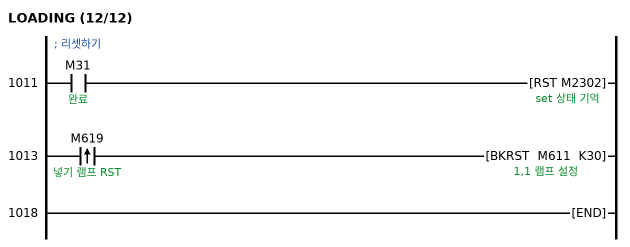
[picture p24: ladder of LOADING, rungs at steps 1011 to 1018]
; 리셋하기
1011  LD      M31  ; 완료
      RST     M2302  ; set 상태 기억
1013  LDP     M619  ; 넣기 램프 RST
      BKRST   M611 K30  ; 1,1 램프 설정
1018  END
END_PROGRAM

PROGRAM UNLOAD
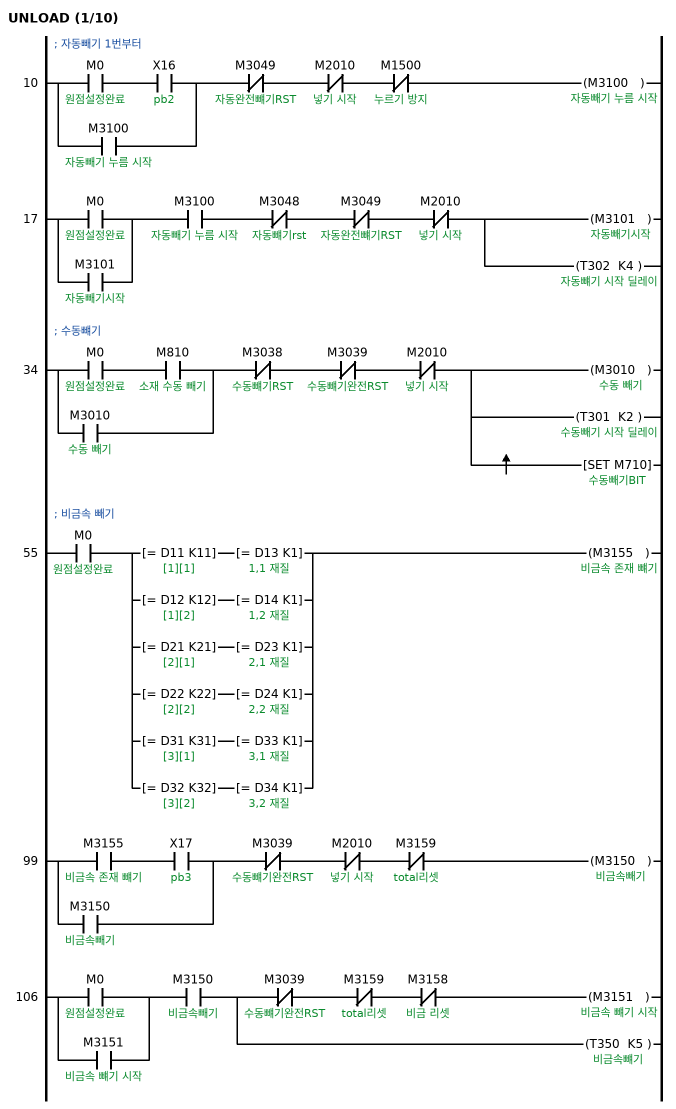
; 자동빼기 1번부터
10    LD      M0  ; 원점설정완료
      AND     X16  ; pb2
      OR      M3100  ; 자동빼기 누름 시작
      ANI     M3049  ; 자동완전뺴기RST
      ANI     M2010  ; 넣기 시작
      ANI     M1500  ; 누르기 방지
      OUT     M3100  ; 자동빼기 누름 시작
17    LD      M0  ; 원점설정완료
      OR      M3101  ; 자동빼기시작
      AND     M3100  ; 자동빼기 누름 시작
      ANI     M3048  ; 자동뺴기rst
      ANI     M3049  ; 자동완전뺴기RST
      ANI     M2010  ; 넣기 시작
      OUT     M3101  ; 자동빼기시작
      OUT     T302 K4  ; 자동뺴기 시작 딜레이
; 수동뺴기
34    LD      M0  ; 원점설정완료
      AND     M810  ; 소재 수동 빼기
      OR      M3010  ; 수동 빼기
      ANI     M3038  ; 수동뺴기RST
      ANI     M3039  ; 수동뺴기완전RST
      ANI     M2010  ; 넣기 시작
      OUT     M3010  ; 수동 빼기
      OUT     T301 K2  ; 수동빼기 시작 딜레이
      MEP
      SET     M710  ; 수동빼기BIT
; 비금속 빼기
55    LD      M0  ; 원점설정완료
      LD=     D11 K11  ; [1][1]
      AND=    D13 K1  ; 1,1 재질
      LD=     D12 K12  ; [1][2]
      AND=    D14 K1  ; 1,2 재질
      ORB
      LD=     D21 K21  ; [2][1]
      AND=    D23 K1  ; 2,1 재질
      ORB
      LD=     D22 K22  ; [2][2]
      AND=    D24 K1  ; 2,2 재질
      ORB
      LD=     D31 K31  ; [3][1]
      AND=    D33 K1  ; 3,1 재질
      ORB
      LD=     D32 K32  ; [3][2]
      AND=    D34 K1  ; 3,2 재질
      ORB
      ANB
      OUT     M3155  ; 비금속 존재 뺴기
99    LD      M3155  ; 비금속 존재 뺴기
      AND     X17  ; pb3
      OR      M3150  ; 비금속빼기
      ANI     M3039  ; 수동뺴기완전RST
      ANI     M2010  ; 넣기 시작
      ANI     M3159  ; total리셋
      OUT     M3150  ; 비금속빼기
106   LD      M0  ; 원점설정완료
      OR      M3151  ; 비금속 뺴기 시작
      AND     M3150  ; 비금속빼기
      MPS
      ANI     M3039  ; 수동뺴기완전RST
      ANI     M3159  ; total리셋
      ANI     M3158  ; 비금 리셋
      OUT     M3151  ; 비금속 뺴기 시작
      MPP
      OUT     T350 K5  ; 비금속뺴기
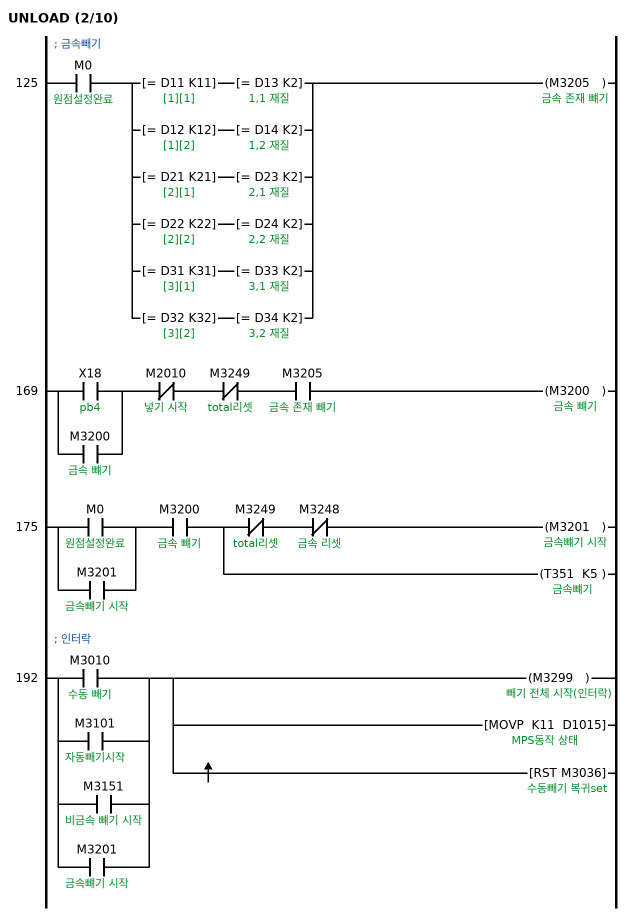
; 금속빼기
125   LD      M0  ; 원점설정완료
      LD=     D11 K11  ; [1][1]
      AND=    D13 K2  ; 1,1 재질
      LD=     D12 K12  ; [1][2]
      AND=    D14 K2  ; 1,2 재질
      ORB
      LD=     D21 K21  ; [2][1]
      AND=    D23 K2  ; 2,1 재질
      ORB
      LD=     D22 K22  ; [2][2]
      AND=    D24 K2  ; 2,2 재질
      ORB
      LD=     D31 K31  ; [3][1]
      AND=    D33 K2  ; 3,1 재질
      ORB
      LD=     D32 K32  ; [3][2]
      AND=    D34 K2  ; 3,2 재질
      ORB
      ANB
      OUT     M3205  ; 금속 존재 뺴기
169   LD      X18  ; pb4
      OR      M3200  ; 금속 뺴기
      ANI     M2010  ; 넣기 시작
      ANI     M3249  ; total리셋
      AND     M3205  ; 금속 존재 뺴기
      OUT     M3200  ; 금속 뺴기
175   LD      M0  ; 원점설정완료
      OR      M3201  ; 금속뺴기 시작
      AND     M3200  ; 금속 뺴기
      MPS
      ANI     M3249  ; total리셋
      ANI     M3248  ; 금속 리셋
      OUT     M3201  ; 금속뺴기 시작
      MPP
      OUT     T351 K5  ; 금속뺴기
; 인터락
192   LD      M3010  ; 수동 빼기
      OR      M3101  ; 자동빼기시작
      OR      M3151  ; 비금속 뺴기 시작
      OR      M3201  ; 금속뺴기 시작
      OUT     M3299  ; 빼기 전체 시작(인터락)
      MOVP    K11 D1015  ; MPS동작 상태
      MEP
      RST     M3036  ; 수동빼기 복귀set
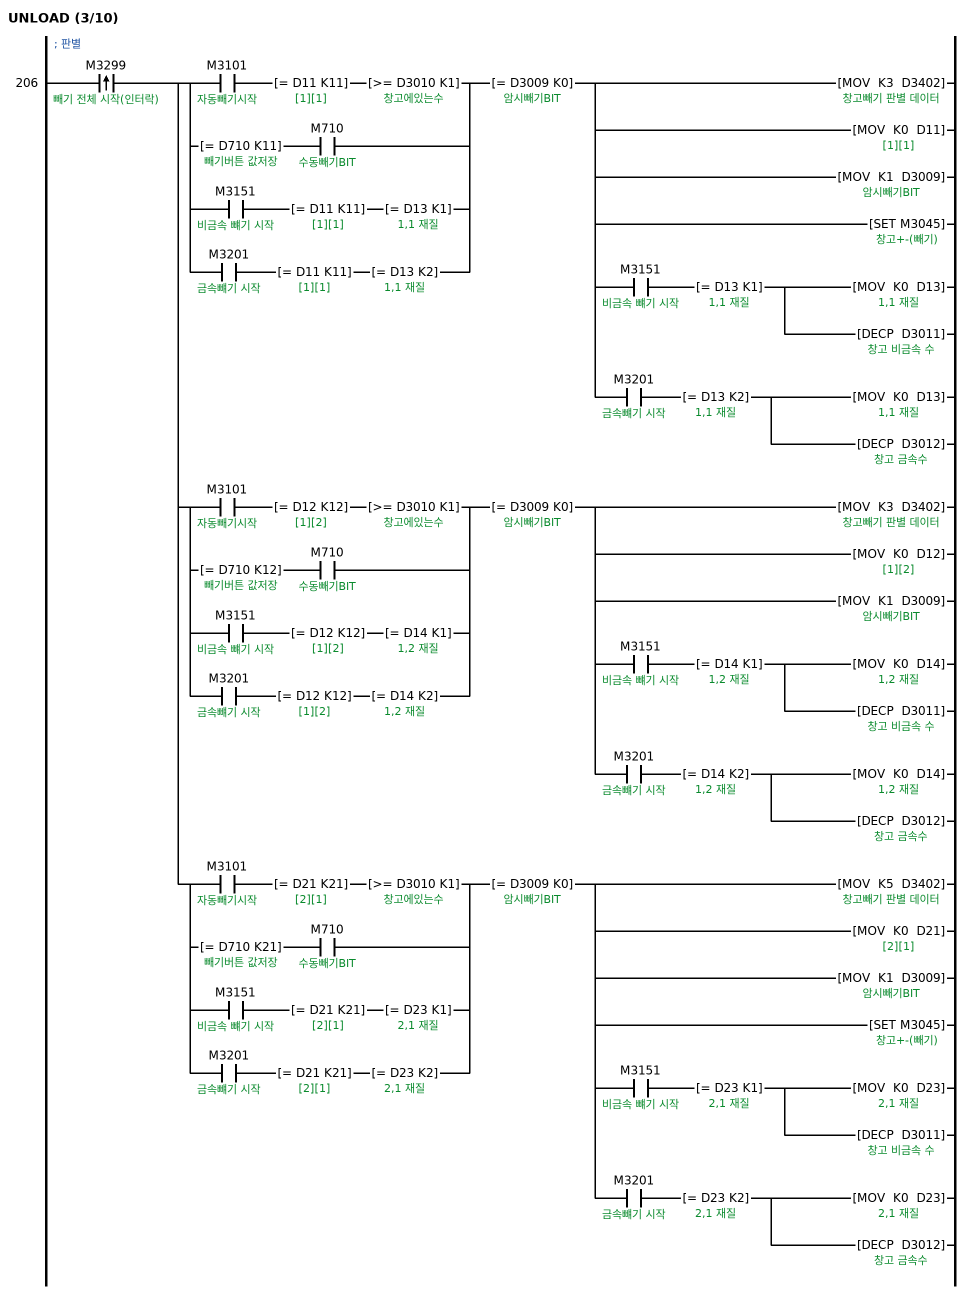
; 판별
206   LDP     M3299  ; 빼기 전체 시작(인터락)
      MPS
      LD      M3101  ; 자동빼기시작
      AND=    D11 K11  ; [1][1]
      AND>=   D3010 K1  ; 창고에있는수
      LD=     D710 K11  ; 빼기버튼 값저장
      AND     M710  ; 수동빼기BIT
      ORB
      LD      M3151  ; 비금속 뺴기 시작
      AND=    D11 K11  ; [1][1]
      AND=    D13 K1  ; 1,1 재질
      ORB
      LD      M3201  ; 금속뺴기 시작
      AND=    D11 K11  ; [1][1]
      AND=    D13 K2  ; 1,1 재질
      ORB
      ANB
      AND=    D3009 K0  ; 암시빼기BIT
      MOV     K3 D3402  ; 창고빼기 판별 데이터
      MOV     K0 D11
      MOV     K1 D3009
      SET     M3045  ; 창고+-(빼기)
      MPS
      AND     M3151  ; 비금속 뺴기 시작
      AND=    D13 K1  ; 1,1 재질
      MOV     K0 D13
      DECP    D3011  ; 창고 비금속 수
      MPP
      AND     M3201  ; 금속뺴기 시작
      AND=    D13 K2  ; 1,1 재질
      MOV     K0 D13
      DECP    D3012  ; 창고 금속수
      MRD
      LD      M3101  ; 자동빼기시작
      AND=    D12 K12  ; [1][2]
      AND>=   D3010 K1  ; 창고에있는수
      LD=     D710 K12  ; 빼기버튼 값저장
      AND     M710  ; 수동빼기BIT
      ORB
      LD      M3151  ; 비금속 뺴기 시작
      AND=    D12 K12  ; [1][2]
      AND=    D14 K1  ; 1,2 재질
      ORB
      LD      M3201  ; 금속뺴기 시작
      AND=    D12 K12  ; [1][2]
      AND=    D14 K2  ; 1,2 재질
      ORB
      ANB
      AND=    D3009 K0  ; 암시빼기BIT
      MOV     K3 D3402
      MOV     K0 D12
      MOV     K1 D3009
      MPS
      AND     M3151  ; 비금속 뺴기 시작
      AND=    D14 K1  ; 1,2 재질
      MOV     K0 D14
      DECP    D3011
      MPP
      AND     M3201  ; 금속뺴기 시작
      AND=    D14 K2  ; 1,2 재질
      MOV     K0 D14
      DECP    D3012
      MPP
      LD      M3101  ; 자동빼기시작
      AND=    D21 K21  ; [2][1]
      AND>=   D3010 K1  ; 창고에있는수
      LD=     D710 K21  ; 빼기버튼 값저장
      AND     M710  ; 수동빼기BIT
      ORB
      LD      M3151  ; 비금속 뺴기 시작
      AND=    D21 K21  ; [2][1]
      AND=    D23 K1  ; 2,1 재질
      ORB
      LD      M3201  ; 금속뺴기 시작
      AND=    D21 K21  ; [2][1]
      AND=    D23 K2  ; 2,1 재질
      ORB
      ANB
      AND=    D3009 K0  ; 암시빼기BIT
      MOV     K5 D3402
      MOV     K0 D21
      MOV     K1 D3009
      SET     M3045  ; 창고+-(빼기)
      MPS
      AND     M3151  ; 비금속 뺴기 시작
      AND=    D23 K1  ; 2,1 재질
      MOV     K0 D23
      DECP    D3011
      MPP
      AND     M3201  ; 금속뺴기 시작
      AND=    D23 K2  ; 2,1 재질
      MOV     K0 D23
      DECP    D3012
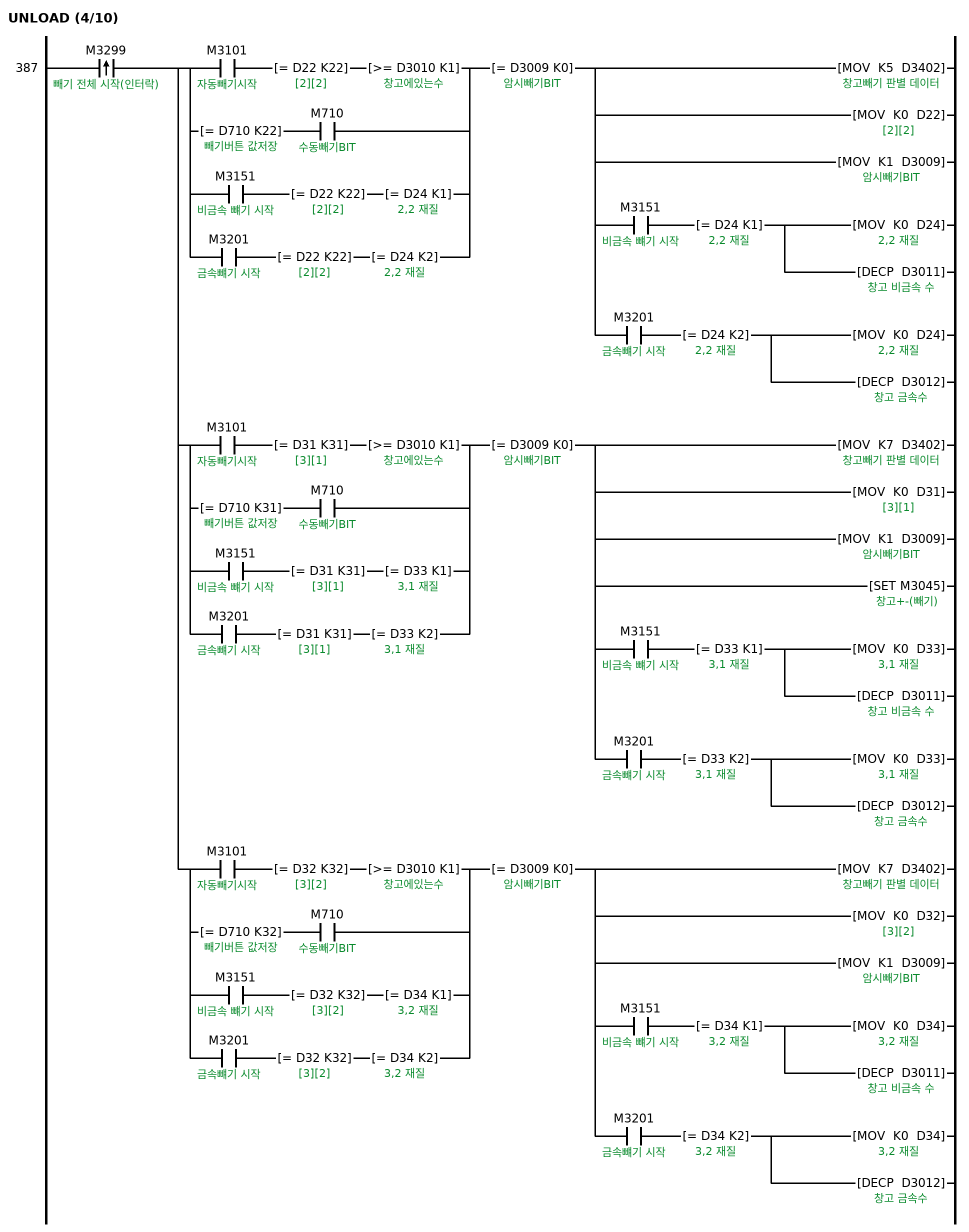
387   LDP     M3299  ; 빼기 전체 시작(인터락)
      MPS
      LD      M3101  ; 자동빼기시작
      AND=    D22 K22  ; [2][2]
      AND>=   D3010 K1  ; 창고에있는수
      LD=     D710 K22  ; 빼기버튼 값저장
      AND     M710  ; 수동빼기BIT
      ORB
      LD      M3151  ; 비금속 뺴기 시작
      AND=    D22 K22  ; [2][2]
      AND=    D24 K1  ; 2,2 재질
      ORB
      LD      M3201  ; 금속뺴기 시작
      AND=    D22 K22  ; [2][2]
      AND=    D24 K2  ; 2,2 재질
      ORB
      ANB
      AND=    D3009 K0  ; 암시빼기BIT
      MOV     K5 D3402
      MOV     K0 D22
      MOV     K1 D3009
      MPS
      AND     M3151  ; 비금속 뺴기 시작
      AND=    D24 K1  ; 2,2 재질
      MOV     K0 D24
      DECP    D3011
      MPP
      AND     M3201  ; 금속뺴기 시작
      AND=    D24 K2  ; 2,2 재질
      MOV     K0 D24
      DECP    D3012
      MRD
      LD      M3101  ; 자동빼기시작
      AND=    D31 K31  ; [3][1]
      AND>=   D3010 K1  ; 창고에있는수
      LD=     D710 K31  ; 빼기버튼 값저장
      AND     M710  ; 수동빼기BIT
      ORB
      LD      M3151  ; 비금속 뺴기 시작
      AND=    D31 K31  ; [3][1]
      AND=    D33 K1  ; 3,1 재질
      ORB
      LD      M3201  ; 금속뺴기 시작
      AND=    D31 K31  ; [3][1]
      AND=    D33 K2  ; 3,1 재질
      ORB
      ANB
      AND=    D3009 K0  ; 암시빼기BIT
      MOV     K7 D3402
      MOV     K0 D31
      MOV     K1 D3009
      SET     M3045  ; 창고+-(빼기)
      MPS
      AND     M3151  ; 비금속 뺴기 시작
      AND=    D33 K1  ; 3,1 재질
      MOV     K0 D33
      DECP    D3011
      MPP
      AND     M3201  ; 금속뺴기 시작
      AND=    D33 K2  ; 3,1 재질
      MOV     K0 D33
      DECP    D3012
      MPP
      LD      M3101  ; 자동빼기시작
      AND=    D32 K32  ; [3][2]
      AND>=   D3010 K1  ; 창고에있는수
      LD=     D710 K32  ; 빼기버튼 값저장
      AND     M710  ; 수동빼기BIT
      ORB
      LD      M3151  ; 비금속 뺴기 시작
      AND=    D32 K32  ; [3][2]
      AND=    D34 K1  ; 3,2 재질
      ORB
      LD      M3201  ; 금속뺴기 시작
      AND=    D32 K32  ; [3][2]
      AND=    D34 K2  ; 3,2 재질
      ORB
      ANB
      AND=    D3009 K0  ; 암시빼기BIT
      MOV     K7 D3402
      MOV     K0 D32
      MOV     K1 D3009
      MPS
      AND     M3151  ; 비금속 뺴기 시작
      AND=    D34 K1  ; 3,2 재질
      MOV     K0 D34
      DECP    D3011
      MPP
      AND     M3201  ; 금속뺴기 시작
      AND=    D34 K2  ; 3,2 재질
      MOV     K0 D34
      DECP    D3012
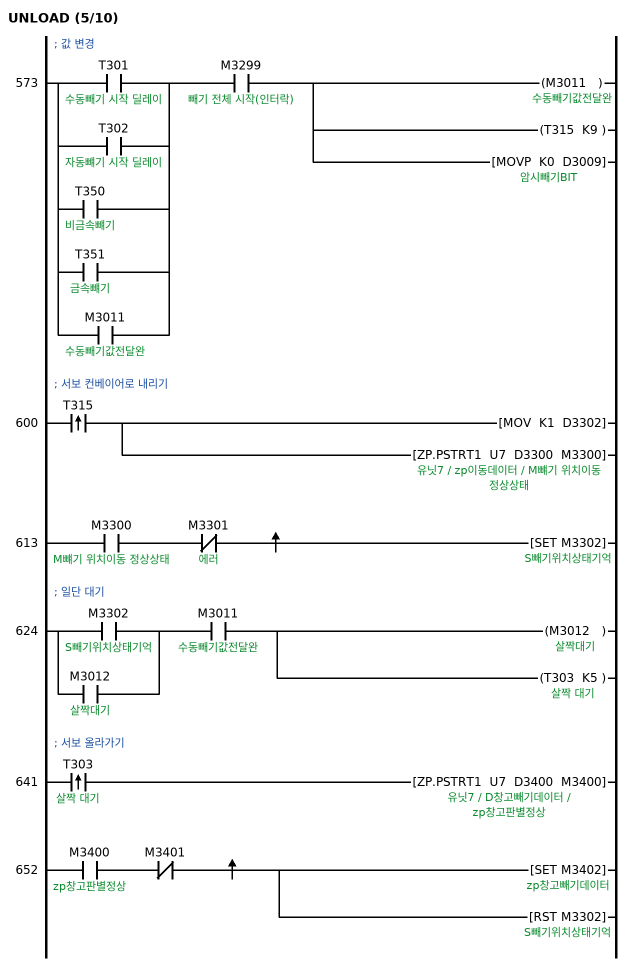
; 값 변경
573   LD      T301  ; 수동빼기 시작 딜레이
      OR      T302  ; 자동뺴기 시작 딜레이
      OR      T350  ; 비금속뺴기
      OR      T351  ; 금속뺴기
      OR      M3011  ; 수동빼기값전달완
      AND     M3299  ; 빼기 전체 시작(인터락)
      OUT     M3011  ; 수동빼기값전달완
      OUT     T315 K9
      MOVP    K0 D3009
; 서보 컨베이어로 내리기
600   LDP     T315
      MOV     K1 D3302
      ZP.PSTRT1 U7 D3300 M3300  ; 유닛7 / zp이동데이터 / M뺴기 위치이동 정상상태
613   LD      M3300  ; M뺴기 위치이동 정상상태
      ANI     M3301  ; 에러
      MEP
      SET     M3302  ; S빼기위치상태기억
; 일단 대기
624   LD      M3302  ; S빼기위치상태기억
      OR      M3012  ; 살짝대기
      AND     M3011  ; 수동빼기값전달완
      OUT     M3012  ; 살짝대기
      OUT     T303 K5  ; 살짝 대기
; 서보 올라가기
641   LDP     T303  ; 살짝 대기
      ZP.PSTRT1 U7 D3400 M3400  ; D창고빼기데이터 / zp창고판별정상
652   LD      M3400  ; zp창고판별정상
      ANI     M3401
      MEP
      SET     M3402  ; zp창고빼기데이터
      RST     M3302  ; S빼기위치상태기억
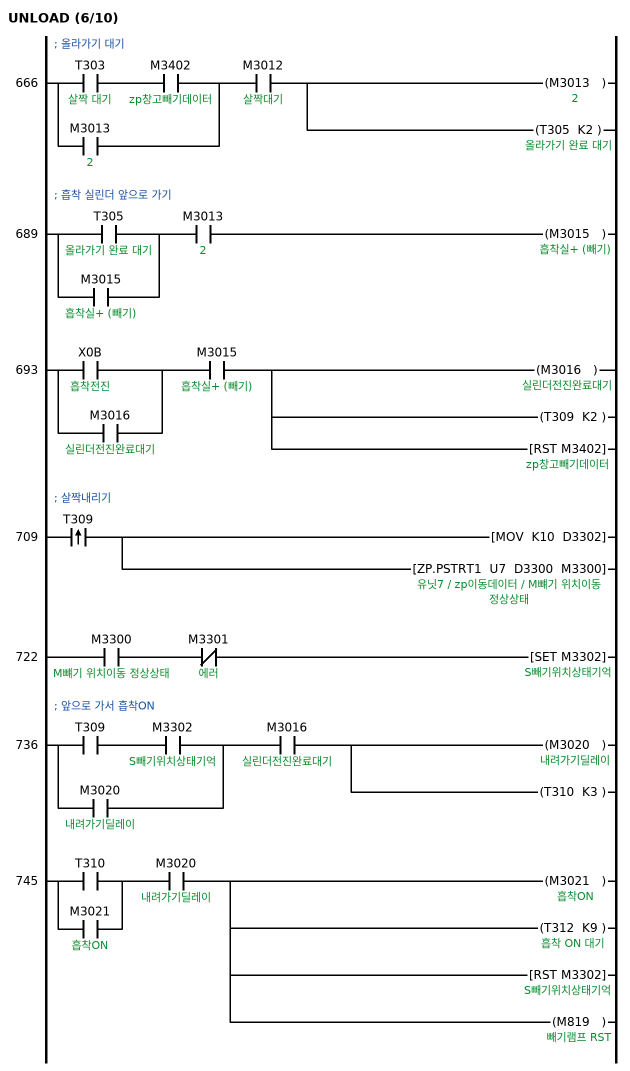
; 올라가기 대기
666   LD      T303  ; 살짝 대기
      AND     M3402  ; zp창고빼기데이터
      OR      M3013  ; 2
      AND     M3012  ; 살짝대기
      OUT     M3013  ; 2
      OUT     T305 K2  ; 올라가기 완료 대기
; 흡착 실린더 앞으로 가기
689   LD      T305  ; 올라가기 완료 대기
      OR      M3015  ; 흡착실+ (빼기)
      AND     M3013  ; 2
      OUT     M3015  ; 흡착실+ (빼기)
693   LD      X0B  ; 흡착전진
      OR      M3016  ; 실린더전진완료대기
      AND     M3015  ; 흡착실+ (빼기)
      OUT     M3016  ; 실린더전진완료대기
      OUT     T309 K2
      RST     M3402  ; zp창고빼기데이터
; 살짝내리기
709   LDP     T309
      MOV     K10 D3302
      ZP.PSTRT1 U7 D3300 M3300
722   LD      M3300  ; M뺴기 위치이동 정상상태
      ANI     M3301  ; 에러
      SET     M3302  ; S빼기위치상태기억
; 앞으로 가서 흡착ON
736   LD      T309
      AND     M3302  ; S빼기위치상태기억
      OR      M3020  ; 내려가기딜레이
      AND     M3016  ; 실린더전진완료대기
      OUT     M3020  ; 내려가기딜레이
      OUT     T310 K3
745   LD      T310
      OR      M3021  ; 흡착ON
      AND     M3020  ; 내려가기딜레이
      OUT     M3021  ; 흡착ON
      OUT     T312 K9  ; 흡착 ON 대기
      RST     M3302  ; S빼기위치상태기억
      OUT     M819  ; 빼기램프 RST
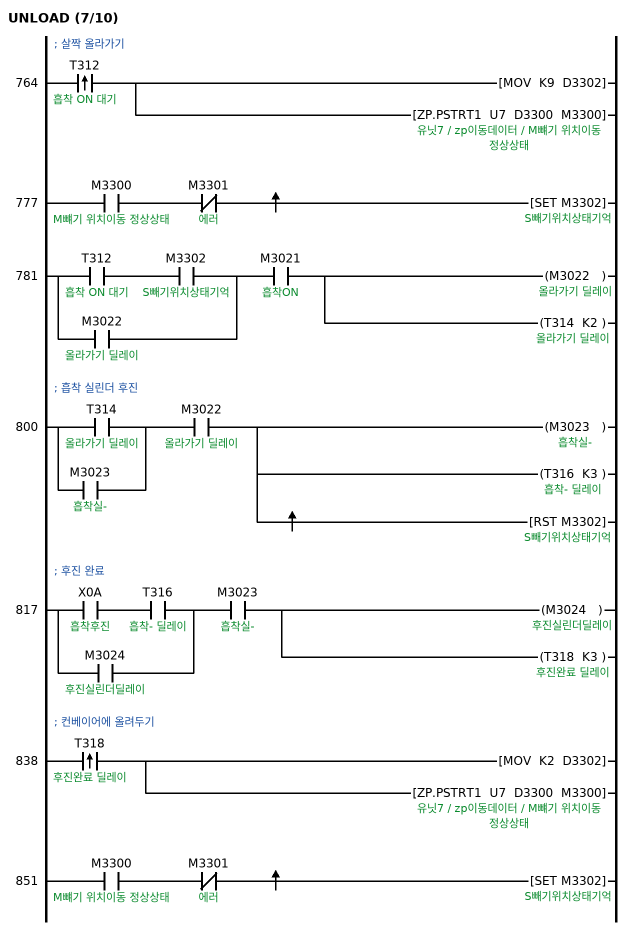
; 살짝 올라가기
764   LDP     T312  ; 흡착 ON 대기
      MOV     K9 D3302
      ZP.PSTRT1 U7 D3300 M3300
777   LD      M3300  ; M뺴기 위치이동 정상상태
      ANI     M3301  ; 에러
      MEP
      SET     M3302  ; S빼기위치상태기억
781   LD      T312  ; 흡착 ON 대기
      AND     M3302  ; S빼기위치상태기억
      OR      M3022  ; 올라가기 딜레이
      AND     M3021  ; 흡착ON
      OUT     M3022  ; 올라가기 딜레이
      OUT     T314 K2  ; 올라가기 딜레이
; 흡착 실린더 후진
800   LD      T314  ; 올라가기 딜레이
      OR      M3023  ; 흡착실-
      AND     M3022  ; 올라가기 딜레이
      OUT     M3023  ; 흡착실-
      OUT     T316 K3  ; 흡착- 딜레이
      MEP
      RST     M3302  ; S빼기위치상태기억
; 후진 완료
817   LD      X0A  ; 흡착후진
      AND     T316  ; 흡착- 딜레이
      OR      M3024  ; 후진실린더딜레이
      AND     M3023  ; 흡착실-
      OUT     M3024  ; 후진실린더딜레이
      OUT     T318 K3  ; 후진완료 딜레이
; 컨베이어에 올려두기
838   LDP     T318  ; 후진완료 딜레이
      MOV     K2 D3302
      ZP.PSTRT1 U7 D3300 M3300
851   LD      M3300  ; M뺴기 위치이동 정상상태
      ANI     M3301  ; 에러
      MEP
      SET     M3302  ; S빼기위치상태기억
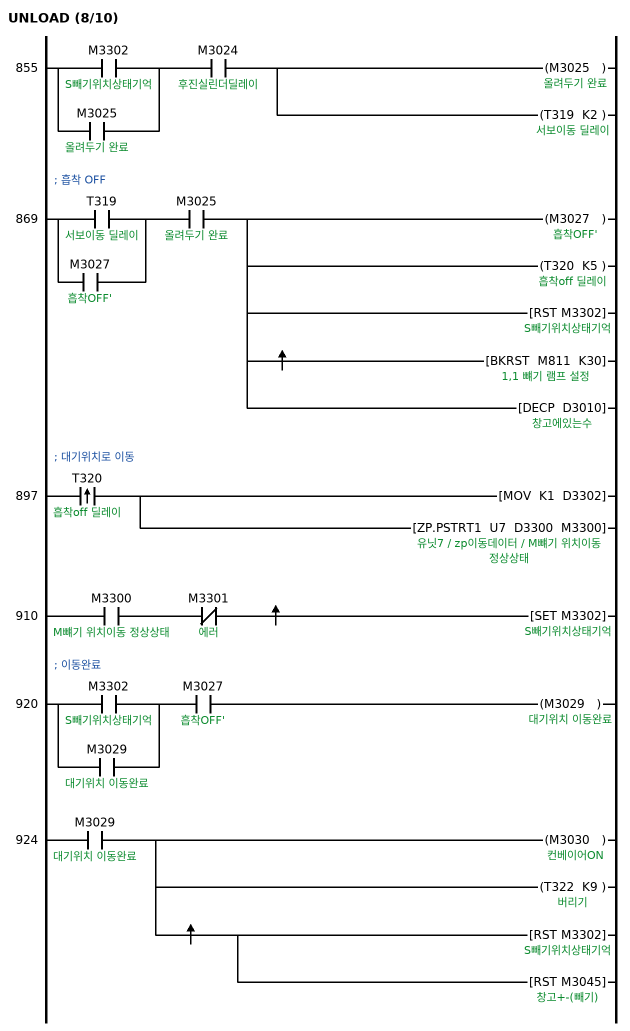
855   LD      M3302  ; S빼기위치상태기억
      OR      M3025  ; 올려두기 완료
      AND     M3024  ; 후진실린더딜레이
      OUT     M3025  ; 올려두기 완료
      OUT     T319 K2  ; 서보이동 딜레이
; 흡착 OFF
869   LD      T319  ; 서보이동 딜레이
      OR      M3027  ; 흡착OFF'
      AND     M3025  ; 올려두기 완료
      OUT     M3027  ; 흡착OFF'
      OUT     T320 K5  ; 흡착off 딜레이
      RST     M3302  ; S빼기위치상태기억
      MPS
      MEP
      BKRST   M811 K30  ; 1,1 뺴기 램프 설정
      MPP
      DECP    D3010
; 대기위치로 이동
897   LDP     T320  ; 흡착off 딜레이
      MOV     K1 D3302
      ZP.PSTRT1 U7 D3300 M3300
910   LD      M3300  ; M뺴기 위치이동 정상상태
      ANI     M3301  ; 에러
      MEP
      SET     M3302  ; S빼기위치상태기억
; 이동완료
920   LD      M3302  ; S빼기위치상태기억
      OR      M3029  ; 대기위치 이동완료
      AND     M3027  ; 흡착OFF'
      OUT     M3029  ; 대기위치 이동완료
924   LD      M3029  ; 대기위치 이동완료
      OUT     M3030  ; 컨베이어ON
      OUT     T322 K9  ; 버리기
      MEP
      RST     M3302  ; S빼기위치상태기억
      RST     M3045  ; 창고+-(빼기)
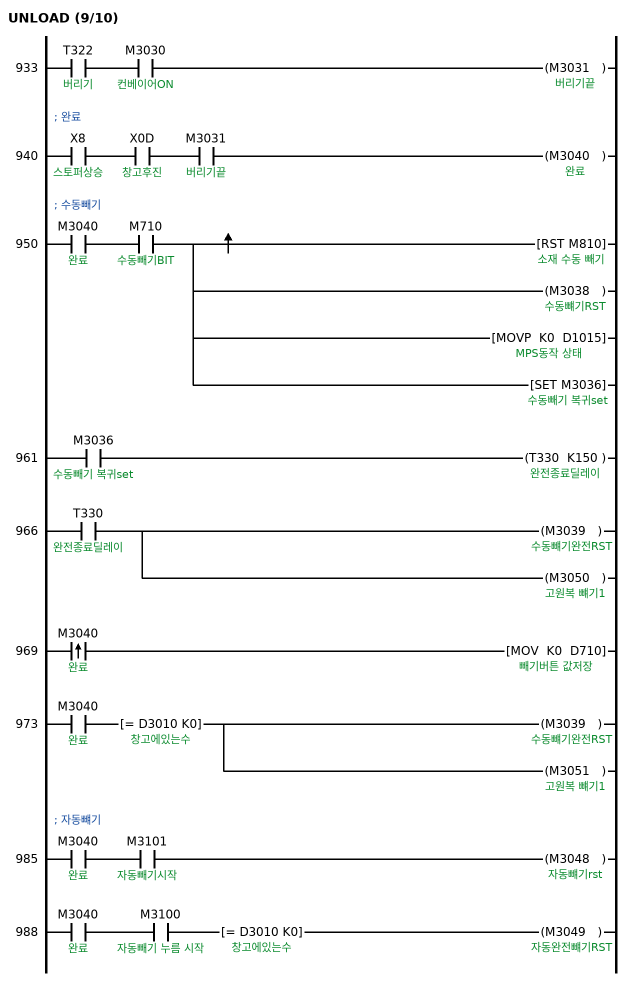
933   LD      T322  ; 버리기
      AND     M3030  ; 컨베이어ON
      OUT     M3031  ; 버리기끝
; 완료
940   LD      X8  ; 스토퍼상승
      AND     X0D  ; 창고후진
      AND     M3031  ; 버리기끝
      OUT     M3040  ; 완료
; 수동빼기
950   LD      M3040  ; 완료
      AND     M710  ; 수동빼기BIT
      MPS
      MEP
      RST     M810  ; 소재 수동 빼기
      MPP
      OUT     M3038  ; 수동뺴기RST
      MOVP    K0 D1015
      SET     M3036  ; 수동빼기 복귀set
961   LD      M3036  ; 수동빼기 복귀set
      OUT     T330 K150  ; 완전종료딜레이
966   LD      T330  ; 완전종료딜레이
      OUT     M3039  ; 수동뺴기완전RST
      OUT     M3050  ; 고원복 뺴기1
969   LDP     M3040  ; 완료
      MOV     K0 D710
973   LD      M3040  ; 완료
      AND=    D3010 K0  ; 창고에있는수
      OUT     M3039  ; 수동뺴기완전RST
      OUT     M3051  ; 고원복 뺴기1
; 자동뺴기
985   LD      M3040  ; 완료
      AND     M3101  ; 자동빼기시작
      OUT     M3048  ; 자동뺴기rst
988   LD      M3040  ; 완료
      AND     M3100  ; 자동빼기 누름 시작
      AND=    D3010 K0  ; 창고에있는수
      OUT     M3049  ; 자동완전뺴기RST
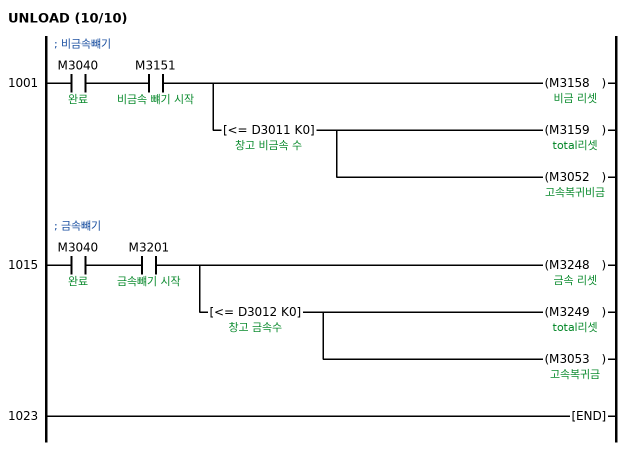
; 비금속뺴기
1001  LD      M3040  ; 완료
      AND     M3151  ; 비금속 뺴기 시작
      OUT     M3158  ; 비금 리셋
      AND<=   D3011 K0  ; 창고 비금속 수
      OUT     M3159  ; total리셋
      OUT     M3052  ; 고속복귀비금
; 금속뺴기
1015  LD      M3040  ; 완료
      AND     M3201  ; 금속뺴기 시작
      OUT     M3248  ; 금속 리셋
      AND<=   D3012 K0  ; 창고 금속수
      OUT     M3249  ; total리셋
      OUT     M3053  ; 고속복귀금
1023  END
END_PROGRAM

PROGRAM MANUAL
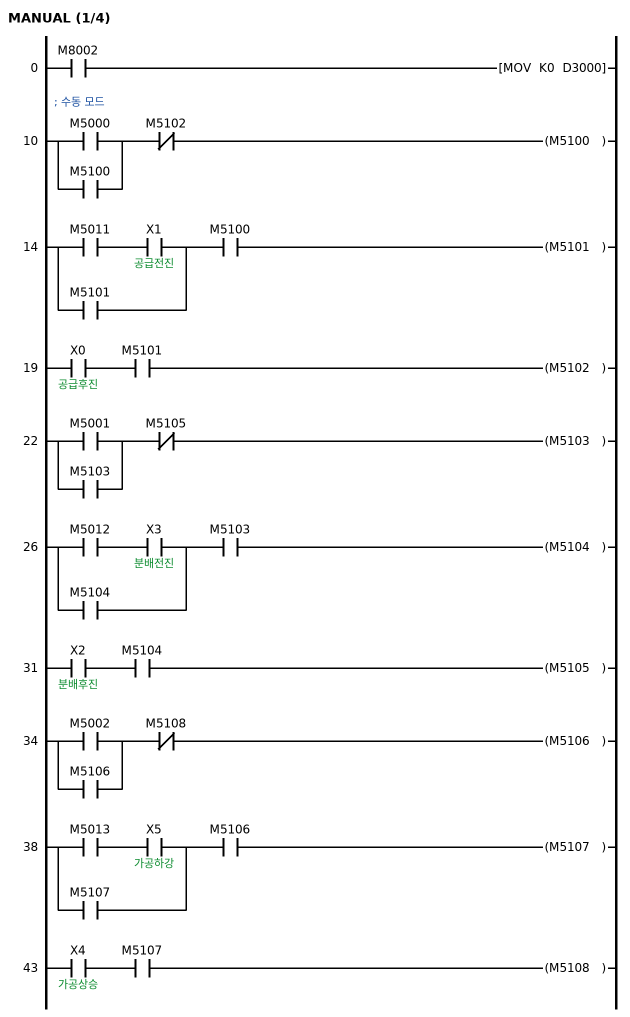
0     LD      M8002
      MOV     K0 D3000
; 수동 모드
10    LD      M5000
      OR      M5100
      ANI     M5102
      OUT     M5100
14    LD      M5011
      AND     X1  ; 공급전진
      OR      M5101
      AND     M5100
      OUT     M5101
19    LD      X0  ; 공급후진
      AND     M5101
      OUT     M5102
22    LD      M5001
      OR      M5103
      ANI     M5105
      OUT     M5103
26    LD      M5012
      AND     X3  ; 분배전진
      OR      M5104
      AND     M5103
      OUT     M5104
31    LD      X2  ; 분배후진
      AND     M5104
      OUT     M5105
34    LD      M5002
      OR      M5106
      ANI     M5108
      OUT     M5106
38    LD      M5013
      AND     X5  ; 가공하강
      OR      M5107
      AND     M5106
      OUT     M5107
43    LD      X4  ; 가공상승
      AND     M5107
      OUT     M5108
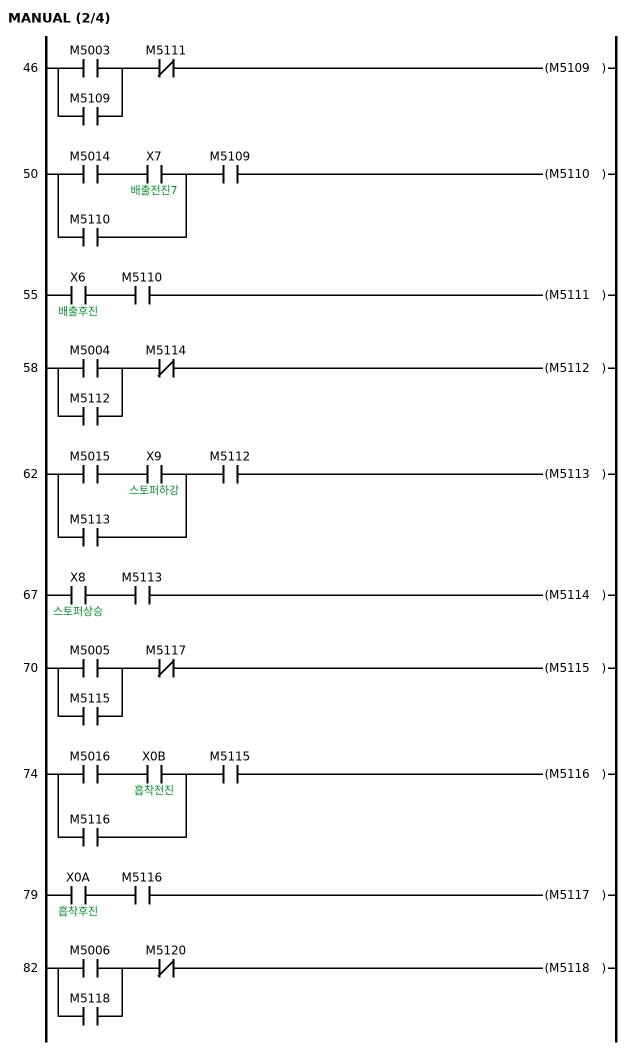
46    LD      M5003
      OR      M5109
      ANI     M5111
      OUT     M5109
50    LD      M5014
      AND     X7  ; 배출전진7
      OR      M5110
      AND     M5109
      OUT     M5110
55    LD      X6  ; 배출후진
      AND     M5110
      OUT     M5111
58    LD      M5004
      OR      M5112
      ANI     M5114
      OUT     M5112
62    LD      M5015
      AND     X9  ; 스토퍼하강
      OR      M5113
      AND     M5112
      OUT     M5113
67    LD      X8  ; 스토퍼상승
      AND     M5113
      OUT     M5114
70    LD      M5005
      OR      M5115
      ANI     M5117
      OUT     M5115
74    LD      M5016
      AND     X0B  ; 흡착전진
      OR      M5116
      AND     M5115
      OUT     M5116
79    LD      X0A  ; 흡착후진
      AND     M5116
      OUT     M5117
82    LD      M5006
      OR      M5118
      ANI     M5120
      OUT     M5118
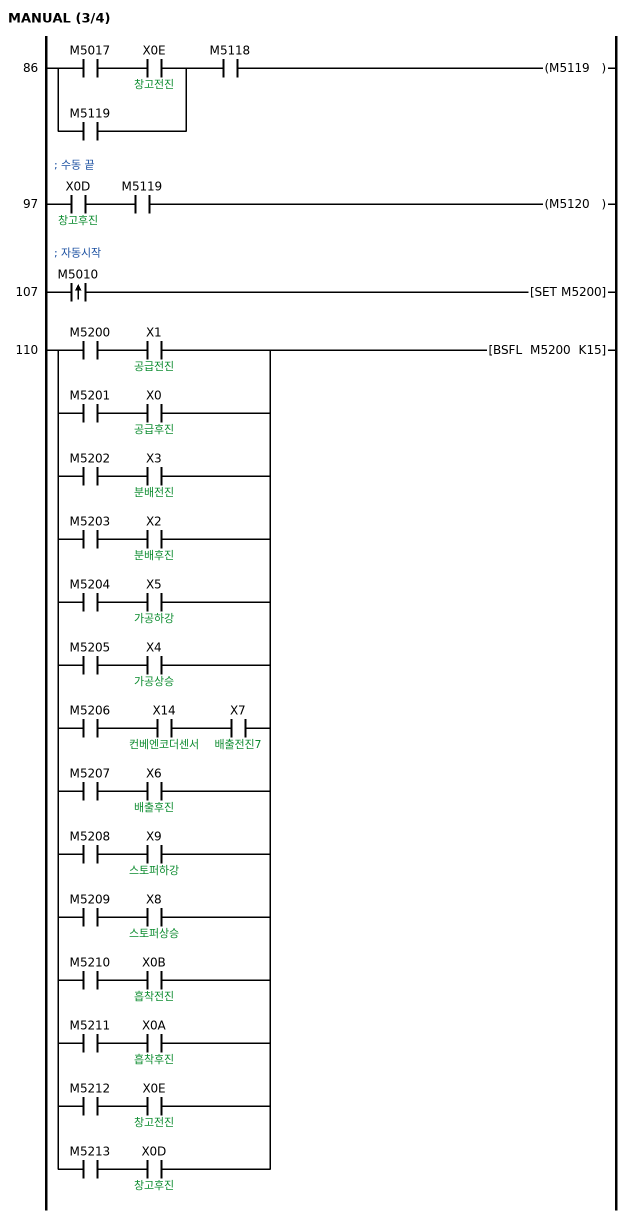
86    LD      M5017
      AND     X0E  ; 창고전진
      OR      M5119
      AND     M5118
      OUT     M5119
; 수동 끝
97    LD      X0D  ; 창고후진
      AND     M5119
      OUT     M5120
; 자동시작
107   LDP     M5010
      SET     M5200
110   LD      M5200
      AND     X1  ; 공급전진
      LD      M5201
      AND     X0  ; 공급후진
      ORB
      LD      M5202
      AND     X3  ; 분배전진
      ORB
      LD      M5203
      AND     X2  ; 분배후진
      ORB
      LD      M5204
      AND     X5  ; 가공하강
      ORB
      LD      M5205
      AND     X4  ; 가공상승
      ORB
      LD      M5206
      AND     X14  ; 컨베엔코더센서
      AND     X7  ; 배출전진7
      ORB
      LD      M5207
      AND     X6  ; 배출후진
      ORB
      LD      M5208
      AND     X9  ; 스토퍼하강
      ORB
      LD      M5209
      AND     X8  ; 스토퍼상승
      ORB
      LD      M5210
      AND     X0B  ; 흡착전진
      ORB
      LD      M5211
      AND     X0A  ; 흡착후진
      ORB
      LD      M5212
      AND     X0E  ; 창고전진
      ORB
      LD      M5213
      AND     X0D  ; 창고후진
      ORB
      BSFL    M5200 K15
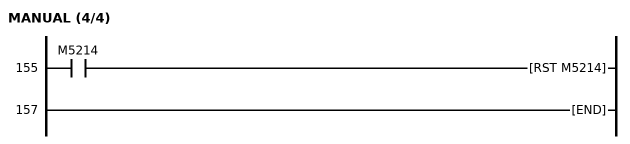
155   LD      M5214
      RST     M5214
157   END
END_PROGRAM

// device comments not shown above
X0C  ; 흡착물건여부
X10  ; 소재센서2
X19  ; pb5
X1A  ; pb6
X1B  ; pb7
X1C  ; toggle
Y30  ; L1
Y31  ; L2
Y32  ; L3
Y33  ; L4
Y34  ; L5
Y35  ; L6
Y36  ; L7
Y80  ; 위결서보
M14  ; 분배+
M23  ; 스토퍼+
M51  ; 배출+
M70  ; 모터ON
M71  ; 가공+
M72  ; 가공-
M73  ; 모터OFF
M74  ; 가공카운터반복
M100  ; 빼기시작
M101  ; 뺴기2
M110  ; 순차뺴기시작
M111  ; 순차2
M198  ; 내부rst
M199  ; 전체리셋
M800  ; 임시 7개이상임
M820  ; 2,1 뺴기 램프 설정
M950  ; 연결
M951  ; 2차연결
M991  ; 내부초기화핗료함
M1006  ; 비상해제
M2041  ; 창고+(비금속)
M2141  ; 창고+ 금속
M2221  ; 창고- (비금)
M2231  ; 창고-   (금속)
M3149  ; 뺴기연결
T0  ; 공급대기
T22  ; 살짝올라가기
T23  ; 살짝 내려가기
T24  ; 흡착OFF대기
T25  ; 살짝 올라가기
T30  ; 비금속컨베off대기
T31  ; 금속컨베off대가
T71  ; 가공 대기 시간
T227  ; 내려가기 대기
D73  ; 소재 대기시간 초단위
D74  ; 소재 대기시간 나머지
D1010  ; 에러시작
D1020  ; 수량 시작
D1030  ; 시간 시작
D1031  ; 소재 없음 대기 시간
D1033  ; 가공 시간
D1101  ; 완료시 상태
D1320  ; 비금속d
D4009  ; 적재 그래프 개수
C70  ; 가공카운터
